FUNCTION_BLOCK Check_AerateOC_Input (* Basic Function Block Type *)
  (* Standard: 61499-2 *)
  (* Version 0.0, 4/2/2024, SESA371406, Schneider Electric, Template *)
  PACKAGE SE.Nereda;
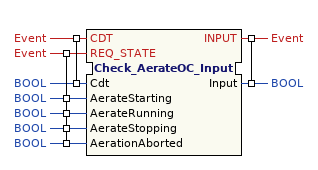
  EVENT_INPUT
    CDT WITH Cdt;
    REQ_STATE WITH AerateStarting, AerateRunning, AerateStopping, AerationAborted;
  END_EVENT
  EVENT_OUTPUT
    INPUT WITH Input;
  END_EVENT
  VAR_INPUT
    Cdt : BOOL;
    AerateStarting : BOOL;
    AerateRunning : BOOL;
    AerateStopping : BOOL;
    AerationAborted : BOOL;
  END_VAR
  VAR_OUTPUT
    Input : BOOL;
  END_VAR
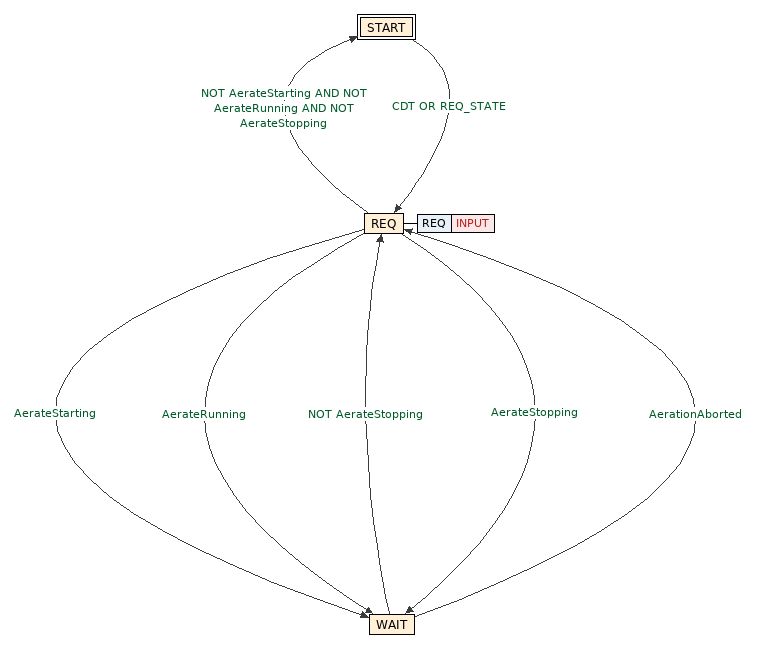
  EC_STATES
    START; (* Initial State *)
    REQ : REQ -> INPUT; (* Normal execution *)
    WAIT;
  END_STATES
  EC_TRANSITIONS
    START TO REQ := CDT  OR REQ_STATE;
    REQ TO START := NOT AerateStarting AND NOT AerateRunning AND NOT AerateStopping;
    REQ TO WAIT := AerateStarting;
    WAIT TO REQ := NOT AerateStopping;
    REQ TO WAIT := AerateRunning;
    REQ TO WAIT := AerateStopping;
    WAIT TO REQ := AerationAborted;
  END_TRANSITIONS
  ALGORITHM REQ IN ST: (* Normally executed algorithm *)
;

IF NOT (Cdt AND NOT(AerateStarting OR AerateRunning OR AerateStopping)) THEN
	Input := TRUE;
ELSE
	Input := FALSE;
END_IF;
  END_ALGORITHM
END_FUNCTION_BLOCK
